FUNCTION_BLOCK TYPE_CONVERTER_1I_11B (* Composite Function Block Type *)
  (* Standard: 61499-2 *)
  (* Version 1.0, 2019-04-02, adeel *)
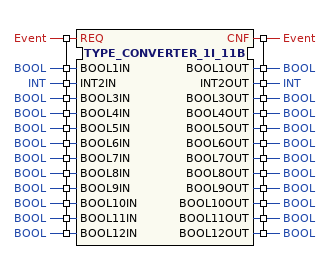
  EVENT_INPUT
    REQ WITH BOOL1IN, INT2IN, BOOL3IN, BOOL4IN, BOOL5IN, BOOL6IN, BOOL7IN, BOOL8IN, BOOL9IN, BOOL10IN, BOOL11IN, BOOL12IN; (* Normal Execution Request *)
  END_EVENT
  EVENT_OUTPUT
    CNF WITH BOOL1OUT, INT2OUT, BOOL3OUT, BOOL4OUT, BOOL5OUT, BOOL6OUT, BOOL7OUT, BOOL8OUT, BOOL9OUT, BOOL10OUT, BOOL11OUT, BOOL12OUT; (* Execution Confirmation *)
  END_EVENT
  VAR_INPUT
    BOOL1IN : BOOL;
    INT2IN : INT;
    BOOL3IN : BOOL;
    BOOL4IN : BOOL;
    BOOL5IN : BOOL;
    BOOL6IN : BOOL;
    BOOL7IN : BOOL;
    BOOL8IN : BOOL;
    BOOL9IN : BOOL;
    BOOL10IN : BOOL;
    BOOL11IN : BOOL;
    BOOL12IN : BOOL;
  END_VAR
  VAR_OUTPUT
    BOOL1OUT : BOOL;
    INT2OUT : INT;
    BOOL3OUT : BOOL;
    BOOL4OUT : BOOL;
    BOOL5OUT : BOOL;
    BOOL6OUT : BOOL;
    BOOL7OUT : BOOL;
    BOOL8OUT : BOOL;
    BOOL9OUT : BOOL;
    BOOL10OUT : BOOL;
    BOOL11OUT : BOOL;
    BOOL12OUT : BOOL;
  END_VAR
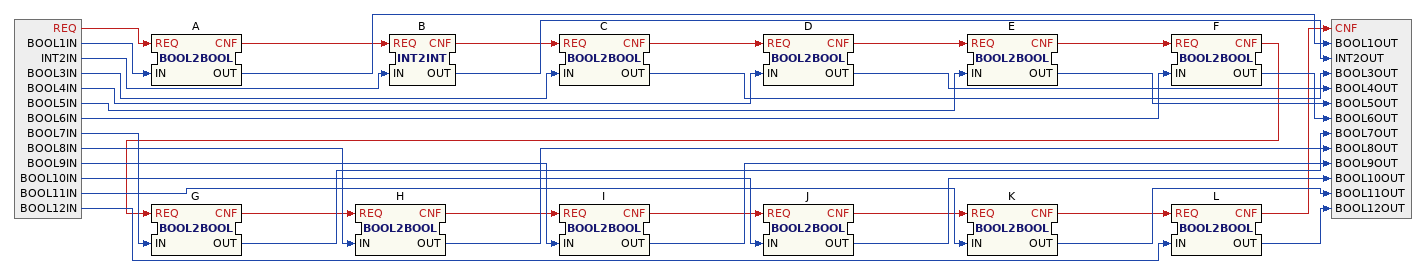
  FBS
    B : INT2INT;
    G : BOOL2BOOL;
    H : BOOL2BOOL;
    I : BOOL2BOOL;
    J : BOOL2BOOL;
    K : BOOL2BOOL;
    L : BOOL2BOOL;
    E : BOOL2BOOL;
    F : BOOL2BOOL;
    A : BOOL2BOOL;
    C : BOOL2BOOL;
    D : BOOL2BOOL;
  END_FBS
  EVENT_CONNECTIONS
    REQ TO A.REQ;
    A.CNF TO B.REQ;
    B.CNF TO C.REQ;
    C.CNF TO D.REQ;
    D.CNF TO E.REQ;
    E.CNF TO F.REQ;
    F.CNF TO G.REQ;
    G.CNF TO H.REQ;
    H.CNF TO I.REQ;
    I.CNF TO J.REQ;
    J.CNF TO K.REQ;
    K.CNF TO L.REQ;
    L.CNF TO CNF;
  END_CONNECTIONS
  DATA_CONNECTIONS
    INT2IN TO B.IN;
    B.OUT TO INT2OUT;
    BOOL1IN TO A.IN;
    BOOL3IN TO C.IN;
    BOOL4IN TO D.IN;
    BOOL5IN TO E.IN;
    BOOL6IN TO F.IN;
    BOOL7IN TO G.IN;
    BOOL8IN TO H.IN;
    BOOL9IN TO I.IN;
    BOOL10IN TO J.IN;
    BOOL11IN TO K.IN;
    BOOL12IN TO L.IN;
    A.OUT TO BOOL1OUT;
    C.OUT TO BOOL3OUT;
    D.OUT TO BOOL4OUT;
    E.OUT TO BOOL5OUT;
    F.OUT TO BOOL6OUT;
    G.OUT TO BOOL7OUT;
    H.OUT TO BOOL8OUT;
    I.OUT TO BOOL9OUT;
    J.OUT TO BOOL10OUT;
    K.OUT TO BOOL11OUT;
    L.OUT TO BOOL12OUT;
  END_CONNECTIONS
END_FUNCTION_BLOCK
